Fanuc KAREL source: kt00731.KL

-- PROVISIONAL review KL for V1013-1; original PC SHA256 b90345e1dc3d28617b915400148cc6694f623f6a140174443c7ae8e6229d7628
-- Incomplete behavior may be omitted. Consult companion uncertainty JSON. Do not deploy.
PROGRAM KT00731
%NOLOCKGROUP
VAR
  OUT : INTEGER
-- UNRESOLVED_DECL ARG type=002010
BEGIN
  -- UNRESOLVED_PC offsets 5-18; opcodes 22,1D,23
  -- UNRESOLVED_PC offsets 23-27; opcodes 7F
END KT00731
